{attribute 'qualified_only'}
{attribute 'strict'}
TYPE eP_calculateMode :
(
	Affine := 0,
	Homography := 1
);
END_TYPE

(* stored: Version 1.1.0.1, ProductVersion 3.1.4024.11
   DUT eP_calculateMode: Id {e7da2a45-ded9-467a-9059-85e7cbbd8b06} *)
